FUNCTION_BLOCK LinearAirPiston EXTENDS AirPiston IMPLEMENTS I_LinearContinuousDrive
VAR_INPUT
	sensorDefaultState : BOOL;
END_VAR
VAR
	homingComplete : BOOL;
	
	home AT %I* : BOOL;
	extendLimit AT %I* : BOOL;
	
	step : Homing;
END_VAR

SUPER^();

override();

PROPERTY AtExtendLimit : BOOL
GET
AtExtendLimit := extendLimit <> sensorDefaultState;
END_GET
END_PROPERTY

{attribute 'monitoring':='call'}
PROPERTY AtHome : BOOL
GET
AtHome := home <> sensorDefaultState;
END_GET
END_PROPERTY

{attribute 'monitoring':='call'}
PROPERTY HomeSet : BOOL
GET
HomeSet := homingComplete;
END_GET
END_PROPERTY

METHOD homingSequence : BOOL
(*
homing sequence is different for linear motion devices with limit sensors
*)
CASE step OF
	Homing.IDLE:
		reset();
		IF bEnable THEN
			step := Homing.START;
		END_IF
		
	Homing.START:
		IF AtHome THEN
			step := Homing.STOP;
			
		ELSIF AtExtendLimit THEN
			step := Homing.RETRY;
			
		ELSE
			moveContinuous(newDirection:= MC_Positive_Direction);
		END_IF
		
	Homing.STOP:
		IF stop() THEN
			step := Homing.DONE;
		END_IF
		
	Homing.DONE:
		homingComplete := TRUE;
		step := Homing.IDLE;
		
END_CASE
END_METHOD

METHOD PROTECTED override : BOOL
VAR_INPUT
END_VAR
IF
	(AtHome AND valveRetract) OR
	(AtExtendLimit AND valveExtend)
THEN
	stop();
END_IF
END_METHOD

END_FUNCTION_BLOCK

(* stored: Version 1.1.0.1, ProductVersion 3.1.4024.11
   POU LinearAirPiston: Id {3cef2aa2-5619-40e9-a961-d9bddd8851a4}, SpecialFunc None
   Folder Properties: Id {cd6ecf69-0a0b-4417-a89f-1a96b349c02e}
   Property AtExtendLimit: Id {1f931d61-2087-4e1f-b43e-e22deeef294a}
   Get Get: Id {29e861d5-7e9e-4f52-8d8c-5175648613b8}
   Property AtHome: Id {7bd78f61-fc51-4fc6-be1e-257cd072f0a4}
   Get Get: Id {13482ca2-7a67-4c1d-b5b9-a9c44f4b97ef}
   Property HomeSet: Id {a58908be-c4d2-4f47-ac47-0ce758f783fe}
   Get Get: Id {c9b261b1-c9ef-428e-817c-3b1579a88dcd}
   Method homingSequence: Id {bd498af7-ec09-4bac-b5ee-2364ab0e9ed8}
   Method override: Id {0ca8edcb-acdf-4fec-90f5-556f8d6a55b7} *)
